FUNCTION_BLOCK LinearServoNC EXTENDS ServoNC IMPLEMENTS I_LinearEncodedDrive
VAR_INPUT
	sensorDefaultState : BOOL;
	
	homeAt0 : BOOL;
	allowDualSideTraverse : BOOL; //allows motion between home to retractLimit
END_VAR
VAR
	homePosition : LREAL;
	extendLimitPosition : LREAL;
	
	homingComplete : BOOL;
	
	home AT %I* : BOOL;
	extendLimit AT %I* : BOOL;
	retractLimit AT %I* : BOOL;
	
	step : Homing;
END_VAR

PROPERTY AtExtendLimit : BOOL
GET
AtExtendLimit := extendLimit <> sensorDefaultState;
END_GET
END_PROPERTY

{attribute 'monitoring':='call'}
PROPERTY AtHome : BOOL
GET
AtHome := home <> sensorDefaultState;
END_GET
END_PROPERTY

PROPERTY AtRetractLimit : BOOL
GET
AtRetractLimit := retractLimit <> sensorDefaultState;
END_GET
END_PROPERTY

{attribute 'monitoring':='call'}
PROPERTY HomeSet : BOOL
GET
HomeSet := homingComplete;
END_GET
END_PROPERTY

METHOD homingSequence : BOOL
(*
homing sequence is different for linear motion devices with limit sensors
*)
CASE step OF
	Homing.IDLE:
		reset();
		IF bEnable THEN
			step := Homing.RETRY;
		END_IF
		
	Homing.START:
		IF AtHome THEN
			step := Homing.STOP;
			
		ELSIF AtRetractLimit THEN
			step := Homing.RETRY;
			
		ELSE
			moveContinuous(newDirection:= MC_Positive_Direction);
		END_IF
		
	Homing.RETRY:
		IF AtExtendLimit THEN
			step := Homing.START;
		ELSE
			moveContinuous(newDirection:= MC_Positive_Direction);
		END_IF
		
	Homing.STOP:
		IF stop() THEN
			step := Homing.SET;
		END_IF
		
	Homing.SET:
		IF CurrentPosition = 0 THEN
			step := Homing.DONE;
		ELSE
			setPosition(newPosition := 0);
		END_IF
		
	Homing.DONE:
		homingComplete := TRUE;
		step := Homing.IDLE;
		
END_CASE
END_METHOD

METHOD PROTECTED override : BOOL
VAR_INPUT
END_VAR
IF
	(AtRetractLimit AND velocity > 0) OR
	(NOT allowDualSideTraverse AND AtHome AND velocity > 0) OR
	(AtExtendLimit AND velocity < 0)
THEN
	stop();
END_IF
END_METHOD

METHOD toHome : BOOL
VAR_INPUT
END_VAR
moveAbsolute(newTarget := 0);
END_METHOD

END_FUNCTION_BLOCK

(* stored: Version 1.1.0.1, ProductVersion 3.1.4024.11
   POU LinearServoNC: Id {ca6375cb-1a16-4775-bbd3-f77de2f39f3e}, SpecialFunc None
   Folder Properties: Id {1c09a678-5067-478d-9089-fff161c6d496}
   Property AtExtendLimit: Id {e51070bb-9c2c-4abf-8149-efdabd42d235}
   Get Get: Id {9444760d-d911-45e6-83b5-1c5cf5f5a8d3}
   Property AtHome: Id {a999cbbf-fb5f-4fdc-9608-5c52bb6de6f3}
   Get Get: Id {fc664c1d-24de-4de6-a350-8223397b54bf}
   Property AtRetractLimit: Id {745d1c76-1804-4a97-aebb-dacd772e9d8b}
   Get Get: Id {6f946ff4-0e20-4a60-9ec4-bf27e7a31a18}
   Property HomeSet: Id {abb6f94c-3735-4a24-8612-4a6fdb76b3aa}
   Get Get: Id {ab64dd72-aea0-4867-9bde-6be2cda4d7f4}
   Method homingSequence: Id {ede81edf-0797-42a0-9d24-d66a2d477cdf}
   Method override: Id {afa3921e-e05c-4dfb-b71d-9a40ed77ae34}
   Method toHome: Id {062630e5-4fda-487e-b35c-caa87684c14b} *)
